PROGRAM P_MitsubishiCommunication
VAR
	i								:INT;
	j								:INT;

	bTwinCATRun						AT %Q* :BOOL;		//三菱のX2に入力
	bTwinCATModbusStart				AT %Q* :BOOL;		//三菱のX3に入力
	bTwinCATAlarm					AT %Q* :BOOL;		//三菱のx4に入力
	bMitsubishiRun					AT %I* :BOOL;		//三菱のY4より出力
	bMitsubishiModbusStart			AT %I* :BOOL;		//三菱のY5より出力	
	bMitsubishiAlarm				AT %I* :BOOL;		//三菱のY6より出力
	
	bMitsubishiModbusOK				: BOOL;
	
	uliCountSpeed					:ULINT;
	
	fbTonBlink1						:ton;
	fbTonBlink2						:ton;
	tBlinkTine						:TIME:=T#130MS;
	
	fbTonRunCheck1					:ton;
	fbTonRunCheck2					:ton;
	
	fbTonMcPower					:ton;
	fbMcPowerREdge					:R_TRIG;
	fbMcPowerFEdge					:F_TRIG;
	
	testes							:ARRAY[1..30] OF REAL;

END_VAR

//-----三菱へ出力-----
	bTwinCATModbusStart:=TRUE;
	bTwinCATRun:=TRUE;
	
	IF GVL.eMachineState < E_MachineState.Stay THEN
		bTwinCATAlarm:=FALSE;
	ELSE
		bTwinCATAlarm:=TRUE;
	END_IF

//---三菱より入力---
	IF bMitsubishiRun=FALSE THEN
		RETURN;
	ELSIF bMitsubishiModbusStart=FALSE THEN
		RETURN;
	ELSIF GVL.mb_Output_Coils[8]=TRUE THEN
		GVL.stAlarm[E_AlarmList.MITSUBISHIAlarm].bFlag:=FALSE;
		GVL.stAlarm[E_AlarmList.MITSUBISHIAlarm].eMachineStateSet:=E_MachineState.Base;
	ELSIF bMitsubishiAlarm=FALSE THEN
		GVL.stAlarm[E_AlarmList.MITSUBISHIAlarm].bFlag:=TRUE;
		GVL.stAlarm[E_AlarmList.MITSUBISHIAlarm].eMachineStateSet:=E_MachineState.Warning;
	END_IF

//-----応答速度確認-----
	IF GVL.mb_Input_Coils[14]=TRUE AND GVL.mb_Output_Coils[14]=FALSE THEN;
		uliCountSpeed:=uliCountSpeed+1;
	END_IF

	GVL.mb_Input_Coils[15]:=GVL.mb_Output_Coils[15];//三菱へ応答


//-----三菱にBeckhoff通信中ブリンクで通知-----
	fbTonBlink1(IN:=NOT fbTonBlink2.Q,PT:=tBlinkTine,Q=>fbTonBlink2.IN,ET=>);

	GVL.mb_Input_Coils[0]:=fbTonBlink1.Q;

	fbTonBlink2(IN:=,PT:=tBlinkTine,Q=>,ET=>);


//-----三菱シーケンサ通信中確認-----
	fbTonRunCheck1(IN:=GVL.mb_Output_Coils[0],PT:=T#500MS,Q=>,ET=>);
	fbTonRunCheck2(IN:=NOT GVL.mb_Output_Coils[0],PT:=T#500MS,Q=>,ET=>);
	
	bMitsubishiModbusOK:=fbTonRunCheck1.Q OR fbTonRunCheck2.Q;


//-----McPoerのOnとOff------
	fbMcPowerREdge(CLK:=GVL.mb_Output_Coils[4],Q=>);
	fbMcPowerFEdge(CLK:=GVL.mb_Input_Coils[4],Q=>);
	fbTonMcPower(IN:=GVL.mb_Output_Coils[4],PT:=T#3S,Q=>,ET=>);

	IF GVL.bPower=FALSE AND fbMcPowerREdge.Q=TRUE THEN;
		GVL.bPower:=TRUE;
	ELSIF GVL.bPower=TRUE AND fbTonMcPower.Q=TRUE THEN ;
		GVL.bPower:=FALSE;
	ELSIF fbMcPowerFEdge.Q=TRUE THEN;
		GVL.bPower:=FALSE;
	END_IF;
	
	IF GVL.bMcPowerStatus[E_Axis.X_Axis]=TRUE AND GVL.bMcPowerStatus[E_Axis.Y_Axis]=TRUE AND GVL.bMcPowerStatus[E_Axis.Z_Axis]=TRUE AND GVL.bMcPowerStatus[E_Axis.Gripper]=TRUE THEN;
		GVL.mb_Input_Coils[4]:=TRUE;
	ELSE;
		GVL.mb_Input_Coils[4]:=FALSE;
	END_IF;


//-----ゼロポジション実行-----
	IF GVL.mb_Input_Coils[4]=TRUE THEN;
		GVL.bHome:=GVL.mb_Output_Coils[5];
	END_IF

	IF GVL.stMoveHomingOut[E_Axis.X_Axis].Busy=TRUE OR GVL.stMoveHomingOut[E_Axis.Y_Axis].Busy=TRUE OR GVL.stMoveHomingOut[E_Axis.Z_Axis].Busy=TRUE OR GVL.stMoveHomingOut[E_Axis.Gripper].Busy=TRUE THEN;
		GVL.mb_Input_Coils[5]:=TRUE;
	ELSE;
		GVL.mb_Input_Coils[5]:=FALSE;
	END_IF;


//-----Jog実行-----
	IF GVL.mb_Input_Coils[4]=TRUE THEN;
		//X軸
		GVL.bJog[E_Axis.X_Axis]:=GVL.mb_Output_Coils[16];
		GVL.lrJogPosition[E_Axis.X_Axis]:=GVL.mb_Output_Registers[16];
		
		//Y軸
		GVL.bJog[E_Axis.Y_Axis]:=GVL.mb_Output_Coils[17];
		GVL.lrJogPosition[E_Axis.Y_Axis]:=GVL.mb_Output_Registers[17];
		
		//Z軸 ステージにグリッパーがあたるのでZ軸は300無しで
		GVL.bJog[E_Axis.Z_Axis]:=GVL.mb_Output_Coils[18];
		GVL.lrJogPosition[E_Axis.Z_Axis]:=GVL.mb_Output_Registers[18];
		IF GVL.lrJogPosition[E_Axis.Z_Axis]>230 THEN;
			GVL.lrJogPosition[E_Axis.Z_Axis]:=225;
		END_IF

		//グリッパー
		GVL.bJog[E_Axis.Gripper]:=GVL.mb_Output_Coils[19];
		GVL.lrJogPosition[E_Axis.Gripper]:=WORD_TO_INT(GVL.mb_Output_Registers[19]);
	END_IF


//-----停止ボタン----
	IF GVL.mb_Input_Coils[4]=TRUE THEN;
		GVL.bHalt:=GVL.mb_Output_Coils[6];
	END_IF

	

//-----非常停止ボタン-----
	IF GVL.mb_Input_Coils[4]=TRUE THEN;
		GVL.bStop:=NOT GVL.mb_Output_Coils[1];
	END_IF


//-----カメラシャッター応答-----
	GVL.mb_Input_Coils[7]:=GVL.mb_Output_Coils[7];

//-----アラームリセット応答-----
	GVL.mb_Input_Coils[8]:=GVL.mb_Output_Coils[8];

//-----セーフティー非常停止リセット応答-----
	GVL.mb_Input_Coils[9]:=GVL.mb_Output_Coils[9];

	
//-----TEST-----
	IF GVL.mb_Output_Coils[30]=TRUE THEN;
		FOR i := 1 TO 30 BY 1 DO;
			testes[i]:=GVL.mb_Output_Registers[29+i];
		END_FOR
		j:=j+1;
		GVL.mb_Input_Coils[30]:=TRUE;
	ELSE;
		GVL.mb_Input_Coils[30]:=FALSE;
	END_IF

END_PROGRAM

(* stored: Version 1.1.0.1, ProductVersion 3.1.4024.12
   POU P_MitsubishiCommunication: Id {7551431c-0546-4892-8591-c118fe27ff05}, SpecialFunc None *)
